FUNCTION_BLOCK FB_HotEndControl
VAR_INPUT
	setpointTmperature: UINT;
END_VAR
VAR_OUTPUT
	done: BOOL;
END_VAR
VAR
	HotEndTemperature: DINT;
	Error: DINT;
END_VAR

END_FUNCTION_BLOCK

(* stored: Version 1.1.0.1, ProductVersion 3.1.4024.9
   POU FB_HotEndControl: Id {c588df39-556d-4122-b746-545f88a1c4f1}, SpecialFunc None *)
